// TIA Portal V18 export
FUNCTION "SS1_IOupdate" : Void   // FC11000, LAD
{ S7_Optimized_Access := 'TRUE' }
VERSION : 0.1
// stored: AutoNumber false, IsIECCheckEnabled false, SetENOAutomatically false, UDAEnableTagReadback false
BEGIN

REGION Network 1
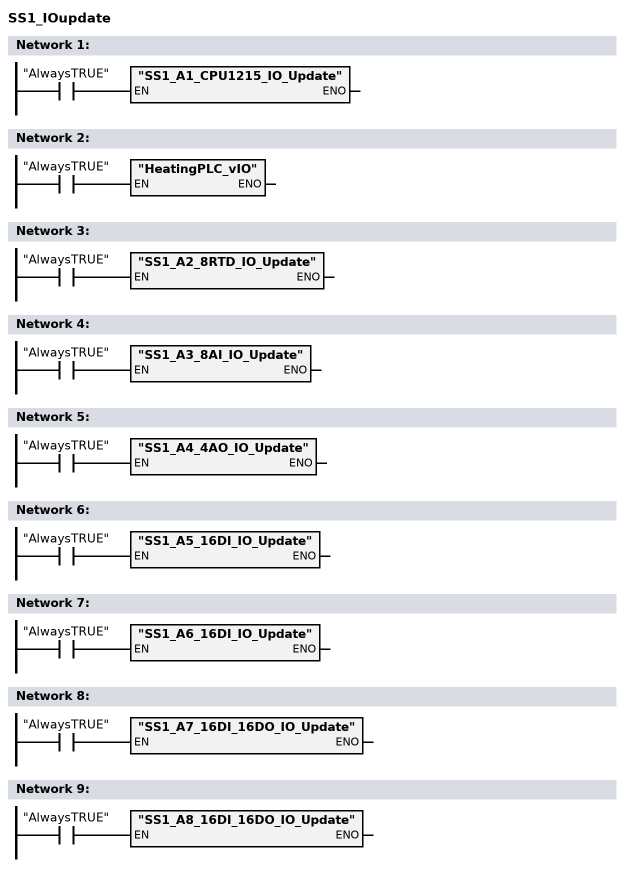
   RUNG wire#powerrail
      Contact( "AlwaysTRUE" )
      "SS1_A1_CPU1215_IO_Update"()
   END_RUNG
   // the same network as SCL:
   IF "AlwaysTRUE" THEN "SS1_A1_CPU1215_IO_Update"(); END_IF;
END_REGION

REGION Network 2
   RUNG wire#powerrail
      Contact( "AlwaysTRUE" )
      "HeatingPLC_vIO"()
   END_RUNG
   // the same network as SCL:
   IF "AlwaysTRUE" THEN "HeatingPLC_vIO"(); END_IF;
END_REGION

REGION Network 3
   RUNG wire#powerrail
      Contact( "AlwaysTRUE" )
      "SS1_A2_8RTD_IO_Update"()
   END_RUNG
   // the same network as SCL:
   IF "AlwaysTRUE" THEN "SS1_A2_8RTD_IO_Update"(); END_IF;
END_REGION

REGION Network 4
   RUNG wire#powerrail
      Contact( "AlwaysTRUE" )
      "SS1_A3_8AI_IO_Update"()
   END_RUNG
   // the same network as SCL:
   IF "AlwaysTRUE" THEN "SS1_A3_8AI_IO_Update"(); END_IF;
END_REGION

REGION Network 5
   RUNG wire#powerrail
      Contact( "AlwaysTRUE" )
      "SS1_A4_4AO_IO_Update"()
   END_RUNG
   // the same network as SCL:
   IF "AlwaysTRUE" THEN "SS1_A4_4AO_IO_Update"(); END_IF;
END_REGION

REGION Network 6
   RUNG wire#powerrail
      Contact( "AlwaysTRUE" )
      "SS1_A5_16DI_IO_Update"()
   END_RUNG
   // the same network as SCL:
   IF "AlwaysTRUE" THEN "SS1_A5_16DI_IO_Update"(); END_IF;
END_REGION

REGION Network 7
   RUNG wire#powerrail
      Contact( "AlwaysTRUE" )
      "SS1_A6_16DI_IO_Update"()
   END_RUNG
   // the same network as SCL:
   IF "AlwaysTRUE" THEN "SS1_A6_16DI_IO_Update"(); END_IF;
END_REGION

REGION Network 8
   RUNG wire#powerrail
      Contact( "AlwaysTRUE" )
      "SS1_A7_16DI_16DO_IO_Update"()
   END_RUNG
   // the same network as SCL:
   IF "AlwaysTRUE" THEN "SS1_A7_16DI_16DO_IO_Update"(); END_IF;
END_REGION

REGION Network 9
   RUNG wire#powerrail
      Contact( "AlwaysTRUE" )
      "SS1_A8_16DI_16DO_IO_Update"()
   END_RUNG
   // the same network as SCL:
   IF "AlwaysTRUE" THEN "SS1_A8_16DI_16DO_IO_Update"(); END_IF;
END_REGION
END_FUNCTION
